FUNCTION_BLOCK PUBLISH_ED_INT (* Service Interface Function Block Type *)
  (* Standard: 61499-2 *)
  (* Version 0.0, 9/14/2008, Horst Mayer, nxtControl GmbH, template *)
  PACKAGE IEC61499;
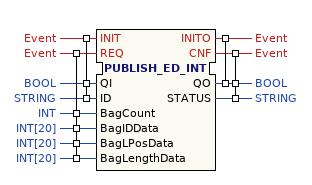
  EVENT_INPUT
    INIT WITH QI, ID;
    REQ WITH BagCount, BagIDData, BagLPosData, BagLengthData;
  END_EVENT
  EVENT_OUTPUT
    INITO WITH QO;
    CNF WITH QO, STATUS;
  END_EVENT
  VAR_INPUT
    QI : BOOL;
    ID : STRING;
    BagCount : INT;
    BagIDData : ARRAY [0..19] OF INT;
    BagLPosData : ARRAY [0..19] OF INT;
    BagLengthData : ARRAY [0..19] OF INT;
  END_VAR
  VAR_OUTPUT
    QO : BOOL; (* Event Output Qualifier *)
    STATUS : STRING;
  END_VAR
END_FUNCTION_BLOCK
